SUBAPPLICATION logiBUS_AI_Raw_Publish_OPC (* logiBUS_AI_IDA (Analog-Eingang) rein Rohwert lesen + per OPC-UA publizieren (DWORD 0-4095), OHNE jegliche VT-Interaktion. Fuer Sensoren, deren physischer Analog-Eingang auf einer Station OHNE VT-Anschluss sitzt (z.B. Hangausgleich-Winkelsensor B14 auf APIXON STG3) - die Kalibrierung + VT-Taster/-Anzeigen laufen dann auf der Station mit VT-Anschluss, gespeist per Remote-Subscribe dieses Rohwerts (siehe logiBUS_AI_Calibrate_3P_Remote_IDA_OPC). *)
  (* Standard: 61499-2; Description: Copyright (c) 2026 Meisterschulen am Ostbahnhof This program and the accompanying materials are made available under the terms of the Eclipse Public License 2.0 which is available at https://www.eclipse.org/legal/epl-2.0/ SPDX-License-Identifier: EPL-2.0 *)
  (* Version 1.0, 2026-09-11, Franz Höpfinger, Meisterschulen am Ostbahnhof, initial implementation - Rohwert-Haelfte von logiBUS_AI_Calibrate_3P_IDA_OPC, fuer Sensoren auf einer Station ohne VT-Anschluss (z.B. Hangausgleich B14 auf STG3). *)
  PACKAGE MyLib::sys;
  IMPORT logiBUS::io::AI::logiBUS_AI;
  IMPORT logiBUS::io::AI::logiBUS_AI_S;
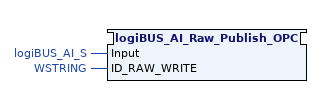
  VAR_INPUT
    Input : logiBUS::io::AI::logiBUS_AI_S := logiBUS_AI::Invalid; (* Identify the Input AnalogInput_I1..I8 *)
    ID_RAW_WRITE : WSTRING; (* Rohwert-Publish-Adresse (DWORD 0-4095, ACTION=PUBLISH), lokal auf dieser Station *)
  END_VAR
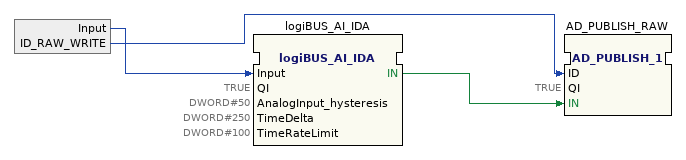
  FBS
    logiBUS_AI_IDA : logiBUS::io::AI::logiBUS_AI_IDA(QI := TRUE, AnalogInput_hysteresis := DWORD#50, TimeDelta := DWORD#250, TimeRateLimit := DWORD#100);
    AD_PUBLISH_RAW : adapter::net::AD_PUBLISH_1(QI := TRUE);
  END_FBS
  DATA_CONNECTIONS
    Input TO logiBUS_AI_IDA.Input;
    ID_RAW_WRITE TO AD_PUBLISH_RAW.ID;
  END_CONNECTIONS
  ADAPTER_CONNECTIONS
    logiBUS_AI_IDA.IN TO AD_PUBLISH_RAW.IN;
  END_CONNECTIONS
END_SUBAPPLICATION
